PROGRAM MAIN
VAR
	toto : BOOL;
END_VAR

toto := NOT toto;

END_PROGRAM

(* stored: Version 1.1.0.1, ProductVersion 3.1.4024.11
   POU MAIN: Id {1a4896df-f497-49c3-94ec-91bd7519a090}, SpecialFunc None *)
